// TIA Portal V19 export
TYPE "C401_VAR_RSS_TYPIC"
   STRUCT
      OBS { ExternalAccessible := 'False'; ExternalVisible := 'False'; ExternalWritable := 'False'} : USInt;   // Observeerbaarheid
      LUS_STO { ExternalAccessible := 'False'; ExternalVisible := 'False'; ExternalWritable := 'False'} : USInt;   // Storingsstatus luspaar
   END_STRUCT;
END_TYPE
